KUKA KRL program: ENABLE_IMPEDANCE.src

&ACCESS RVO1
&REL 8
DEFFCT BOOL ENABLE_IMPEDANCE( )

$STIFFNESS.STRATEGY = 20
$STIFFNESS.COMMIT = TRUE

RETURN TRUE

ENDFCT
